{attribute 'reflection'}
FUNCTION_BLOCK INTERNAL FINAL FB_RPC_Tests EXTENDS TcUnit.FB_TestSuite
VAR
	{attribute 'instance-path'} 
    {attribute 'noinit'} 
	sTestName			: T_MaxString;
	sActiveStep			: T_MaxString;
	nSequence			: INT;
	nSeqOld				: INT;
	nRpcMethodInvoked 	: UDINT;
	aSUTs				: ARRAY[0..255] OF I_RpcReleaseHandle;
END_VAR
VAR_TEMP
	eMode	: E_Mode;
END_VAR

CASE nSequence OF
	0:
		TEST(sTestName);
		F_IncrementStep(nStepToInc:= nSequence, sActiveStep:= sActiveStep, eMode:= E_Mode.INC);
	1:
		sActiveStep := 'ShouldInvokeMethod_NoArguments_NoReturnValue_Successfully';
		TEST(sActiveStep);
		eMode := ShouldInvokeMethod_NoArguments_NoReturnValue_Successfully();
		F_IncrementStep(nStepToInc:= nSequence, sActiveStep, eMode);
	2:
		sActiveStep := 'ShouldInvokeMethod_NoArguments_ReturnValueBoolean_Successfully';
		TEST(sActiveStep);
		eMode := ShouldInvokeMethod_NoArguments_ReturnValueBoolean_Successfully();
		F_IncrementStep(nStepToInc:= nSequence, sActiveStep, eMode);
	3:	
		sActiveStep := 'ShouldInvokeMethod_OneArgument_NoReturnValue_Successfully';
		TEST(sActiveStep);
		eMode := ShouldInvokeMethod_OneArgument_NoReturnValue_Successfully();
		F_IncrementStep(nStepToInc:= nSequence, sActiveStep, eMode);	
	4:	
		sActiveStep := 'ShouldInvokeMethod_OneArgument_NoReturnValue_Successfully';
		TEST(sActiveStep);
		eMode := ShouldInvokeMethod_OneArgument_NoReturnValue_Successfully();
		F_IncrementStep(nStepToInc:= nSequence, sActiveStep, eMode);	
	5:	
		sActiveStep := 'ShouldInvokeMethod_TwoArguments_ReturnValue_Successfully';
		TEST(sActiveStep);
		eMode := ShouldInvokeMethod_TwoArguments_ReturnValue_Successfully();
		F_IncrementStep(nStepToInc:= nSequence, sActiveStep, eMode);
	6:	
		sActiveStep := 'ShouldInvokeMethod_ThreeArguments_ReturnValue_Successfully';
		TEST(sActiveStep);
		eMode := ShouldInvokeMethod_ThreeArguments_ReturnValue_Successfully();
		F_IncrementStep(nStepToInc:= nSequence, sActiveStep, eMode);		
	7:	
		sActiveStep := 'ShouldInvokeMethod_VarInOutConstant_ReturnValue_Successfully';
		TEST(sActiveStep);
		eMode := ShouldInvokeMethod_VarInOutConstant_ReturnValue_Successfully();
		F_IncrementStep(nStepToInc:= nSequence, sActiveStep, eMode);	
	8:	
		sActiveStep := 'ShouldInvokeMethod_VarOutput_ReturnValue_Successfully';
		TEST(sActiveStep);
		eMode := ShouldInvokeMethod_VarOutput_ReturnValue_Successfully();
		F_IncrementStep(nStepToInc:= nSequence, sActiveStep, eMode);	
	9:	
		sActiveStep := 'ShouldInvokeMethod_TwoVarOutput_ReturnValue_Successfully';
		TEST(sActiveStep);
		eMode := ShouldInvokeMethod_TwoVarOutput_ReturnValue_Successfully();
		F_IncrementStep(nStepToInc:= nSequence, sActiveStep, eMode);	
	10:	
		sActiveStep := 'ShouldInvokeMethod_VarInput_VarInOut_VarOutput_ReturnValue_Successfully';
		TEST(sActiveStep);
		eMode := ShouldInvokeMethod_VarInput_VarInOut_VarOutput_ReturnValue_Successfully();
		F_IncrementStep(nStepToInc:= nSequence, sActiveStep, eMode);		
	11: 
		sActiveStep := 'ShouldReturnError0x705';
		TEST(sActiveStep);
		eMode := ShouldReturnError0x705();
		F_IncrementStep(nStepToInc:= nSequence, sActiveStep, eMode);	
	12: 
		sActiveStep := 'ShouldReturnError0x710';
		TEST(sActiveStep);
		eMode := ShouldReturnError0x710();
		F_IncrementStep(nStepToInc:= nSequence, sActiveStep, eMode);	
	13: 
		sActiveStep := 'ShouldReleaseAllSymbolHandleSuccessfully';
		TEST(sActiveStep);
		eMode := ShouldReleaseAllSymbolHandleSuccessfully();
		F_IncrementStep(nStepToInc:= nSequence, sActiveStep, eMode);	
	ELSE
		TEST_FINISHED_NAMED(sTestName);
END_CASE

IF nSequence <> nSeqOld THEN
	nRpcMethodInvoked := 0;
	nSeqOld := nSequence;
END_IF;

{attribute 'TcRpcEnable'}
METHOD NoParameter_NoReturnValue

nRpcMethodInvoked := nRpcMethodInvoked + 1;
END_METHOD

{attribute 'TcRpcEnable'}
METHOD NoParameter_ReturnValue : BOOL
VAR_INPUT
END_VAR
nRpcMethodInvoked := nRpcMethodInvoked + 1;
NoParameter_ReturnValue := nRpcMethodInvoked > 0;
END_METHOD

{attribute 'TcRpcEnable'}
METHOD OneParameter_NoReturnValue
VAR_INPUT
	nArg1 	: UDINT;
END_VAR
nRpcMethodInvoked := nArg1;
END_METHOD

METHOD Register
VAR_INPUT
	ipRpcReleaseHandle	: I_RpcReleaseHandle;
END_VAR

VAR
	i :UINT;
END_VAR


FOR i:=0 TO 255 DO	
	IF aSUTs[i] = ipRpcReleaseHandle THEN
		EXIT;
	END_IF
	IF aSUTs[i] <> NULL THEN
		CONTINUE;
	END_IF
	
	aSUTs[i] := ipRpcReleaseHandle;
	EXIT;
END_FOR
END_METHOD

METHOD ShouldInvokeMethod_NoArguments_NoReturnValue_Successfully : E_Mode

VAR_INST
	fbSUT		: FB_RPC(GCL.cLocalAmsNetId, _AppInfo.AdsPort, 'PRG_UnitTests.fbRpcTests', 'NoParameter_NoReturnValue');
END_VAR

VAR
	stRetVal	: ST_AdsStatus;
	eMode		: E_Mode := E_MODE.BUSY;
END_VAR
// Arrange
Register(fbSUT);

// Act
stRetVal := fbSUT.Invoke();

IF NOT stRetVal.bBusy THEN
	eMode := E_Mode.INC;
	
	// Assert
	AssertFalse(Condition:= stRetVal.bError, Message:= 'Expected method NoParameter_NoReturnValue to return no error.');
	AssertEquals_UDINT(Expected:= E_AdsErr.NOERR, Actual:= stRetVal.nError, Message:= 'Expected method NoParameter_NoReturnValue to return no error.');
	AssertEquals_UDINT(Expected:= 1, Actual:= nRpcMethodInvoked, Message:= 'Expected method NoParameter_NoReturnValue to be invoked once.');
END_IF

ShouldInvokeMethod_NoArguments_NoReturnValue_Successfully := eMode;
END_METHOD

METHOD ShouldInvokeMethod_NoArguments_ReturnValueBoolean_Successfully : E_Mode

VAR_INST
	fbSUT		: FB_RPC(GCL.cLocalAmsNetId, _AppInfo.AdsPort, 'PRG_UnitTests.fbRpcTests', 'NoParameter_ReturnValue');
END_VAR

VAR
	stRetVal	: ST_AdsStatus;
	eMode		: E_Mode := E_MODE.BUSY;
	bActual		: BOOL;
END_VAR
// Arrange
Register(fbSUT);

// Act
stRetVal := fbSUT.ReturnValue(bActual).Invoke();

IF NOT stRetVal.bBusy THEN
	eMode := E_Mode.INC;
	// Assert
	AssertFalse(Condition:= stRetVal.bError, Message:= 'Expected method NoParameter_ReturnValue to return no error.');
	AssertEquals_UDINT(Expected:= E_AdsErr.NOERR, Actual:= stRetVal.nError, Message:= 'Expected method NoParameter_ReturnValue to return no error.');
	AssertEquals_UDINT(Expected:= 1, Actual:= nRpcMethodInvoked, Message:= 'Expected method NoParameter_ReturnValue to be invoked once.');
	AssertTrue(Condition:= bActual, Message:= 'Expected method NoParameter_ReturnValue to return TRUE.');
END_IF

ShouldInvokeMethod_NoArguments_ReturnValueBoolean_Successfully := eMode;
END_METHOD

METHOD ShouldInvokeMethod_OneArgument_NoReturnValue_Successfully : E_Mode

VAR_INST
	fbSUT		: FB_RPC(GCL.cLocalAmsNetId, _AppInfo.AdsPort, 'PRG_UnitTests.fbRpcTests', 'OneParameter_NoReturnValue');
END_VAR

VAR
	stRetVal	: ST_AdsStatus;
	eMode		: E_Mode := E_MODE.BUSY;
	nArg		: UDINT;
END_VAR
// Arrange
Register(fbSUT);
nArg := 123;

// Act
stRetVal := fbSUT.VarInput(nArg).NoReturnValue().Invoke();

IF NOT stRetVal.bBusy THEN
	eMode := E_Mode.INC;
	
	// Assert
	AssertFalse(Condition:= stRetVal.bError, Message:= 'Expected method OneParameter_NoReturnValue to return no error.');
	AssertEquals_UDINT(Expected:= E_AdsErr.NOERR, Actual:= stRetVal.nError, Message:= 'Expected method OneParameter_NoReturnValue to return no error.');
	AssertEquals_UDINT(Expected:= nArg, Actual:= nRpcMethodInvoked, Message:= 'Expected method OneParameter_NoReturnValue to be invoked with value 123.');
END_IF

ShouldInvokeMethod_OneArgument_NoReturnValue_Successfully := eMode;
END_METHOD

METHOD ShouldInvokeMethod_ThreeArguments_ReturnValue_Successfully : E_Mode

VAR_INST
	fbSUT		: FB_RPC(GCL.cLocalAmsNetId, _AppInfo.AdsPort, 'PRG_UnitTests.fbRpcTests', 'ThreeParameters_ReturnValue');
END_VAR

VAR
	stRetVal	: ST_AdsStatus;
	eMode		: E_Mode := E_MODE.BUSY;
	nArg1		: UDINT;
	stArg2		: ST_AdsStatus;	// IN_OUT!
	sArg3		: STRING;
	sActualRetVal : STRING;
END_VAR
// Arrange
Register(fbSUT);
nArg1 := 456;
stArg2.bBusy := FALSE;
stArg2.bError := TRUE;
stArg2.nError := 321;
sArg3 := 'third Argument';

// Act
stRetVal := fbSUT.VarInput(nArg1).VarInOut(stArg2).VarInput(sArg3).ReturnValue(sActualRetVal).Invoke();

IF NOT stRetVal.bBusy THEN
	eMode := E_Mode.INC;
	
	// Assert
	AssertFalse(Condition:= stRetVal.bError, Message:= 'Expected method TwoParameters_ReturnValue to return no error.');
	AssertEquals_UDINT(Expected:= E_AdsErr.NOERR, Actual:= stRetVal.nError, Message:= 'Expected method ThreeParameters_ReturnValue to return no error.');
	AssertEquals_UDINT(Expected:= nArg1, Actual:= nRpcMethodInvoked, Message:= 'Expected method ThreeParameters_ReturnValue to be invoked with value 456.');
	AssertTrue(Condition:= stArg2.bBusy, Message:= 'Expected method ThreeParameters_ReturnValue to invert bBusy of VAR_IN_OUT');
	AssertFalse(Condition:= stArg2.bError, Message:= 'Expected method ThreeParameters_ReturnValue to invert bError of VAR_IN_OUT');
	AssertEquals_UDINT(Expected:= 321 * 2, Actual:= stArg2.nError, Message:= 'Expected method ThreeParameters_ReturnValue to double value nError of VAR_IN_OUT');
	AssertEquals_STRING(Expected:= sArg3, Actual:= sActualRetVal, Message:= 'Expected method ThreeParameters_ReturnValue to return value .');
END_IF

ShouldInvokeMethod_ThreeArguments_ReturnValue_Successfully := eMode;
END_METHOD

METHOD ShouldInvokeMethod_TwoArguments_ReturnValue_Successfully : E_Mode

VAR_INST
	fbSUT		: FB_RPC(GCL.cLocalAmsNetId, _AppInfo.AdsPort, 'PRG_UnitTests.fbRpcTests', 'TwoParameters_ReturnValue');
END_VAR

VAR
	stRetVal	: ST_AdsStatus;
	eMode		: E_Mode := E_MODE.BUSY;
	nArg1		: UDINT;
	sArg2		: STRING;
	sActualRetVal : STRING;
END_VAR
// Arrange
Register(fbSUT);
nArg1 := 456;
sArg2 := 'second Argument';

// Act
stRetVal := fbSUT.VarInput(nArg1).VarInput(sArg2).ReturnValue(sActualRetVal).Invoke();

IF NOT stRetVal.bBusy THEN
	eMode := E_Mode.INC;
	
	// Assert
	AssertFalse(Condition:= stRetVal.bError, Message:= 'Expected method TwoParameters_ReturnValue to return no error.');
	AssertEquals_UDINT(Expected:= E_AdsErr.NOERR, Actual:= stRetVal.nError, Message:= 'Expected method TwoParameters_ReturnValue to return no error.');
	AssertEquals_UDINT(Expected:= nArg1, Actual:= nRpcMethodInvoked, Message:= 'Expected method TwoParameters_ReturnValue to be invoked with value 456.');
	AssertEquals_STRING(Expected:= sArg2, Actual:= sActualRetVal, Message:= 'Expected method TwoParameters_ReturnValue to return value .');
END_IF

ShouldInvokeMethod_TwoArguments_ReturnValue_Successfully := eMode;
END_METHOD

METHOD ShouldInvokeMethod_TwoVarOutput_ReturnValue_Successfully : E_Mode

VAR_INST
	fbSUT		: FB_RPC(GCL.cLocalAmsNetId, _AppInfo.AdsPort, 'PRG_UnitTests.fbRpcTests', 'TwoVarOutput_ReturnValue');
END_VAR

VAR
	stRetVal	: ST_AdsStatus;
	eMode		: E_Mode := E_MODE.BUSY;
	stArg		: ST_AdsStatus;
	nA			: UDINT;
	nActualRetVal : UDINT;
END_VAR
// Arrange
Register(fbSUT);

// Act
stRetVal := fbSUT.VarOutput(stArg).VarOutput(nA).ReturnValue(nActualRetVal).Invoke();

IF NOT stRetVal.bBusy THEN
	eMode := E_Mode.INC;
	
	// Assert
	AssertFalse(Condition:= stRetVal.bError, Message:= 'Expected method VarOutput_ReturnValue to return no error.');
	AssertEquals_UDINT(Expected:= E_AdsErr.NOERR, Actual:= stRetVal.nError, Message:= 'Expected method VarOutput_ReturnValue to return no error.');
	AssertFalse(Condition:= stArg.bBusy, Message:= 'Expected method VarOutput_ReturnValue to return stArg.bBusy = FALSE');
	AssertTrue(Condition:= stArg.bError, Message:= 'Expected method VarOutput_ReturnValue to return stArg.bError = TRUE');
	AssertEquals_UDINT(Expected:= 123, Actual:= stARg.nError, Message:= 'Expected method VarOutput_ReturnValue to return stArg.nError = 123');
	AssertEquals_UDINT(Expected:= 789, Actual:= nA, Message:= 'Expected method VarOutput_ReturnValue to return nA = 789');
	AssertEquals_UDINT(Expected:= 456, Actual:= nActualRetVal, Message:= 'Expected method VarOutput_ReturnValue to return 456.');
END_IF

ShouldInvokeMethod_TwoVarOutput_ReturnValue_Successfully := eMode;
END_METHOD

METHOD ShouldInvokeMethod_VarInOutConstant_ReturnValue_Successfully : E_Mode

VAR_INST
	fbSUT		: FB_RPC(GCL.cLocalAmsNetId, _AppInfo.AdsPort, 'PRG_UnitTests.fbRpcTests', 'VarInOutConstant_ReturnValue');
END_VAR

VAR
	stRetVal	: ST_AdsStatus;
	eMode		: E_Mode := E_MODE.BUSY;
	stArg		: ST_LibVersion;
	nActualRetVal : UDINT;
END_VAR
// Arrange
Register(fbSUT);
stArg.nFlags := 987;

// Act
stRetVal := fbSUT.VarInOut(stArg).ReturnValue(nActualRetVal).Invoke();

IF NOT stRetVal.bBusy THEN
	eMode := E_Mode.INC;
	
	// Assert
	AssertFalse(Condition:= stRetVal.bError, Message:= 'Expected method VarInOutConstant_ReturnValue to return no error.');
	AssertEquals_UDINT(Expected:= E_AdsErr.NOERR, Actual:= stRetVal.nError, Message:= 'Expected method VarInOutConstant_ReturnValue to return no error.');
	AssertEquals_DWORD(Expected:= 987, Actual:= stArg.nFlags, Message:= 'Expected method VarInOutConstant_ReturnValue to be invoked with value 987.');
	AssertEquals_UDINT(Expected:= 987, Actual:= nActualRetVal, Message:= 'Expected method VarInOutConstant_ReturnValue to be invoked with value 987.');
END_IF

ShouldInvokeMethod_VarInOutConstant_ReturnValue_Successfully := eMode;
END_METHOD

METHOD ShouldInvokeMethod_VarInput_VarInOut_VarOutput_ReturnValue_Successfully : E_Mode

VAR_INST
	fbSUT		: FB_RPC(GCL.cLocalAmsNetId, _AppInfo.AdsPort, 'PRG_UnitTests.fbRpcTests', 'VarInput_VarInOut_VarOutput_ReturnValue');
END_VAR

VAR
	stRetVal	: ST_AdsStatus;
	eMode		: E_Mode := E_MODE.BUSY;
		
	sStrIn		: STRING;
	nIn			: INT;
	nInOut 		: INT;
	stArgOut	: ST_AdsStatus;
	sStrOut		: STRING;	
	sRetVal		: STRING;
END_VAR
// Arrange
Register(fbSUT);

sStrIn	:= 'Input String';
nIn		:= -666;
nInOut	:= 777;

// Act
stRetVal := fbSUT.VarInput(sStrIn).VarInput(nIn).VarInOut(nInOut).VarOutput(stArgOut).VarOutput(sStrOut).ReturnValue(sRetVal).Invoke();

IF NOT stRetVal.bBusy THEN
	eMode := E_Mode.INC;
	
	// Assert
	AssertFalse(Condition:= stRetVal.bError, Message:= 'Expected method VarInput_VarInOut_VarOutput_ReturnValue to return no error.');
	AssertEquals_UDINT(Expected:= E_AdsErr.NOERR, Actual:= stRetVal.nError, Message:= 'Expected method VarInput_VarInOut_VarOutput_ReturnValue to return no error.');
	AssertTrue(Condition:= stArgOut.bBusy, Message:= 'Expected method VarInput_VarInOut_VarOutput_ReturnValue to return stArgOut.bBusy = TRUE');
	AssertFalse(Condition:= stArgOut.bError, Message:= 'Expected method VarInput_VarInOut_VarOutput_ReturnValue to return stArgOut.bError = FALSE');
	AssertEquals_UDINT(Expected:= 222, Actual:= stArgOut.nError, Message:= 'Expected method VarInput_VarInOut_VarOutput_ReturnValue to return stArgOut.nError = 222');
	AssertEquals_STRING(Expected:= 'sStrOut: Input String', Actual:= sStrOut,
						Message:= 'Expected method VarInput_VarInOut_VarOutput_ReturnValue to return "sStrOut: Input String"');
	AssertEquals_STRING(Expected:= 'ReturnValue: Input String', Actual:= sRetVal,
						Message:= 'Expected method VarInput_VarInOut_VarOutput_ReturnValue to return "ReturnValue: Input String"');
END_IF

ShouldInvokeMethod_VarInput_VarInOut_VarOutput_ReturnValue_Successfully := eMode;
END_METHOD

METHOD ShouldInvokeMethod_VarOutput_ReturnValue_Successfully : E_Mode

VAR_INST
	fbSUT		: FB_RPC(GCL.cLocalAmsNetId, _AppInfo.AdsPort, 'PRG_UnitTests.fbRpcTests', 'VarOutput_ReturnValue');
END_VAR

VAR
	stRetVal	: ST_AdsStatus;
	eMode		: E_Mode := E_MODE.BUSY;
	stArg		: ST_AdsStatus;
	nActualRetVal : UDINT;
END_VAR
// Arrange
Register(fbSUT);


// Act
stRetVal := fbSUT.VarOutput(stArg).ReturnValue(nActualRetVal).Invoke();

IF NOT stRetVal.bBusy THEN
	eMode := E_Mode.INC;
	
	// Assert
	AssertFalse(Condition:= stRetVal.bError, Message:= 'Expected method VarOutput_ReturnValue to return no error.');
	AssertEquals_UDINT(Expected:= E_AdsErr.NOERR, Actual:= stRetVal.nError, Message:= 'Expected method VarOutput_ReturnValue to return no error.');
	AssertTrue(Condition:= stArg.bBusy, Message:= 'Expected method VarOutput_ReturnValue to return bBusy = TRUE.');
	AssertFalse(Condition:= stArg.bError, Message:= 'Expected method VarOutput_ReturnValue to return bError = FALSE');
	AssertEquals_UDINT(Expected:= 456, Actual:= stARg.nError, Message:= 'Expected method VarOutput_ReturnValue to return VAR_OUTPUT 456.');
	AssertEquals_UDINT(Expected:= 123, Actual:= nActualRetVal, Message:= 'Expected method VarOutput_ReturnValue to return 123.');
END_IF

ShouldInvokeMethod_VarOutput_ReturnValue_Successfully := eMode;
END_METHOD

METHOD ShouldReleaseAllSymbolHandleSuccessfully : E_Mode

VAR
	stRetVal	: ST_AdsStatus;
	ipSUT		: I_RpcReleaseHandle;
END_VAR

VAR_INST
	nIndex 		: UINT := 0;
END_VAR


ipSUT := aSUTs[nIndex];
IF ipSUT = NULL THEN
	ShouldReleaseAllSymbolHandleSuccessfully := E_Mode.INC;
	RETURN;
END_IF

// Act
stRetVal := ipSUT.ReleaseHandle();

IF NOT stRetVal.bBusy THEN
	nIndex := nIndex + 1;	
	// Assert
	AssertFalse(Condition:= stRetVal.bError, Message:= 'Expected ReleaseHandle to return no error.');
	AssertEquals_UDINT(Expected:= E_AdsErr.NOERR, Actual:= stRetVal.nError, Message:= 'Expected ReleaseHandle to return no error.');
END_IF

ShouldReleaseAllSymbolHandleSuccessfully := E_Mode.BUSY;
END_METHOD

METHOD ShouldReturnError0x705 : E_Mode

VAR_INST
	fbSUT		: FB_RPC(GCL.cLocalAmsNetId, _AppInfo.AdsPort, 'PRG_UnitTests.fbRpcTests', 'NoParameter_NoReturnValue');
END_VAR

VAR
	stRetVal	: ST_AdsStatus;
	eMode		: E_Mode := E_MODE.BUSY;
	nDummy		: INT;
END_VAR
// Act
stRetVal := fbSUT.VarInput(nDummy).NoReturnValue().Invoke();

IF NOT stRetVal.bBusy THEN
	eMode := E_Mode.INC;
	
	// Assert
	AssertTrue(Condition:= stRetVal.bError, Message:= 'Expected method NoParameter_NoReturnValue to return error.');
	AssertEquals_UDINT(Expected:= E_AdsErr.DEVICE_INVALIDSIZE, Actual:= stRetVal.nError, Message:= 'Expected method NoParameter_NoReturnValue to return error ADSERR_DEVICE_INVALIDSIZE.');
	AssertEquals_UDINT(Expected:= 0, Actual:= nRpcMethodInvoked, Message:= 'Expected method NoParameter_NoReturnValue to not be invoked.');
END_IF

ShouldReturnError0x705 := eMode;
END_METHOD

METHOD ShouldReturnError0x710 : E_Mode

VAR_INST
	fbSUT		: FB_RPC(GCL.cLocalAmsNetId, _AppInfo.AdsPort, 'PRG_UnitTests.fbRpcTests', 'NotExistingSymbol');
END_VAR

VAR
	stRetVal	: ST_AdsStatus;
	eMode		: E_Mode := E_MODE.BUSY;
	nDummy		: INT;
END_VAR
// Act
stRetVal := fbSUT.VarInput(nDummy).NoReturnValue().Invoke();

IF NOT stRetVal.bBusy THEN
	eMode := E_Mode.INC;
	
	// Assert
	AssertTrue(Condition:= stRetVal.bError, Message:= 'Expected return error.');
	AssertEquals_UDINT(Expected:= E_AdsErr.DEVICE_SYMBOLNOTFOUND, Actual:= stRetVal.nError, Message:= 'Expected error ADSERR_DEVICE_SYMBOLNOTFOUND.');
END_IF

ShouldReturnError0x710 := eMode;
END_METHOD

{attribute 'TcRpcEnable'}
METHOD ThreeParameters_ReturnValue : STRING
VAR_INPUT
	nArg1 	: UDINT;
END_VAR
VAR_IN_OUT
	stArg2  : ST_AdsStatus;
END_VAR
VAR_INPUT
	sArg3	: STRING;
END_VAR
nRpcMethodInvoked := nArg1;
stArg2.bBusy := NOT stArg2.bBusy;
stArg2.bError := NOT stARg2.bError;
stARg2.nError := stARg2.nError * 2;
ThreeParameters_ReturnValue := sArg3;
END_METHOD

{attribute 'TcRpcEnable'}
METHOD TwoParameters_ReturnValue : STRING
VAR_INPUT
	nArg1 	: UDINT;
	sArg2	: STRING;
END_VAR
nRpcMethodInvoked := nArg1;
TwoParameters_ReturnValue := sArg2;
END_METHOD

{attribute 'TcRpcEnable'}
METHOD TwoVarOutput_ReturnValue : UDINT
VAR_OUTPUT
	stArg	: ST_AdsStatus;
	nA		: UDINT;
END_VAR

stArg.bBusy := FALSE;
stArg.bError := TRUE;
stArg.nError := 123;
nA := 789;
TwoVarOutput_ReturnValue := 456;
END_METHOD

{attribute 'TcRpcEnable'}
METHOD VarInOutConstant_ReturnValue : DWORD
VAR_IN_OUT CONSTANT
	stArg  : ST_LibVersion;
END_VAR
VarInOutConstant_ReturnValue := stArg.nFlags;
END_METHOD

{attribute 'TcRpcEnable'}
METHOD VarInput_VarInOut_VarOutput_ReturnValue : STRING
VAR_INPUT
	sStrIn	: STRING;
	nIn		: INT;
END_VAR
VAR_IN_OUT
	nInOut	: INT;	
END_VAR
VAR_OUTPUT
	stArgOut	: ST_AdsStatus;
	sStrOut 	: STRING;
END_VAR



nInOut := nInOut + nIn;

stArgOut.bBusy := TRUE;
stArgOut.bError := FALSE;
stArgOut.nError := 222;

sStrOut := CONCAT('sStrOut: ',sStrIn);

VarInput_VarInOut_VarOutput_ReturnValue := CONCAT('ReturnValue: ',sStrIn);
END_METHOD

{attribute 'TcRpcEnable'}
METHOD VarOutput_ReturnValue : UDINT
VAR_OUTPUT
	stArg  : ST_AdsStatus;
END_VAR

stArg.bBusy := TRUE;
stArg.bError := FALSE;
stArg.nError := 456;
VarOutput_ReturnValue := 123;
END_METHOD

END_FUNCTION_BLOCK

(* stored: Version 1.1.0.1, ProductVersion 3.1.4024.12
   POU FB_RPC_Tests: Id {cbe11911-4728-435a-ba6b-73a9e68e4ee2}, SpecialFunc None
   Folder Helper: Id {782de686-70f2-40b2-98b5-095d810b423d}
   Folder TestMethods: Id {88b8acb6-f383-4965-aeba-1d77ff91ad95}
   Method NoParameter_NoReturnValue: Id {fe8fa86e-296b-4e40-ab9d-7bf225c643ea}
   Method NoParameter_ReturnValue: Id {5c2a64b3-1c7b-41ce-bcc0-a7635e3f39bc}
   Method OneParameter_NoReturnValue: Id {99590e33-c91a-4294-9383-0dff400e0cd5}
   Method Register: Id {cd0135b3-de6a-46f0-95a5-c26fa1be9a08}
   Method ShouldInvokeMethod_NoArguments_NoReturnValue_Successfully: Id {ebc60a66-099b-4039-aae2-2bdc97f0b383}
   Method ShouldInvokeMethod_NoArguments_ReturnValueBoolean_Successfully: Id {fe09ed6b-dda3-4944-bac3-771b0453401c}
   Method ShouldInvokeMethod_OneArgument_NoReturnValue_Successfully: Id {402c4c52-b3eb-40f7-a68f-1c796a40239a}
   Method ShouldInvokeMethod_ThreeArguments_ReturnValue_Successfully: Id {2a6e6f72-0f5f-414d-80c0-eaa6ccdb3942}
   Method ShouldInvokeMethod_TwoArguments_ReturnValue_Successfully: Id {e1a1bc8c-1ddb-472b-b3c6-bb492613a6f6}
   Method ShouldInvokeMethod_TwoVarOutput_ReturnValue_Successfully: Id {4cc2e689-bef5-4dd4-b6fa-20975d808b8f}
   Method ShouldInvokeMethod_VarInOutConstant_ReturnValue_Successfully: Id {5bb2217d-919f-447d-b86d-337aee153857}
   Method ShouldInvokeMethod_VarInput_VarInOut_VarOutput_ReturnValue_Successfully: Id {24545837-3efd-4197-989a-c9ae6cfefb8e}
   Method ShouldInvokeMethod_VarOutput_ReturnValue_Successfully: Id {9ed56a14-ac2e-4cd5-836f-a35bd8b60b81}
   Method ShouldReleaseAllSymbolHandleSuccessfully: Id {9a28eca6-1d82-498c-92be-b1510e63b3b7}
   Method ShouldReturnError0x705: Id {fcbe1809-94ef-4fc3-8100-ee156ab487ec}
   Method ShouldReturnError0x710: Id {d7a3f3be-7c04-4d09-89b5-a2b705793866}
   Method ThreeParameters_ReturnValue: Id {46ec559a-3fb6-47d8-b43b-5513c26b6c63}
   Method TwoParameters_ReturnValue: Id {dc5d36f9-9a7a-48f8-9ca9-edb900040176}
   Method TwoVarOutput_ReturnValue: Id {653a64de-4ce6-4f1a-9f88-e644ed3a92dd}
   Method VarInOutConstant_ReturnValue: Id {cf312003-3ca4-454c-887f-29a94ca68b7e}
   Method VarInput_VarInOut_VarOutput_ReturnValue: Id {a1d2971b-a107-4ae8-a338-f0a20b0b8707}
   Method VarOutput_ReturnValue: Id {256c405d-d8c7-40b5-9a3f-a81f9b36222e} *)
